// TIA Portal V17 export
// export: Created 2024-08-07T21:44:04.3800599Z, ExportSetting WithDefaults, DisplayName Totally Integrated Automation Portal, DisplayVersion V17 Update 7, DisplayName TIA Portal Openness, DisplayVersion V17 Update 7, DisplayName TIA Portal Version Control Interface, DisplayVersion V17, DisplayName SINAMICS Startdrive Advanced, DisplayVersion V17 SP2, DisplayName SINAMICS Startdrive G110M, G120, G120C, G120D, G120P, G115D, DisplayVersion V17 SP2, DisplayName SINAMICS Startdrive G130, G150, S120, S150, SINAMICS MV, S210, DisplayVersion V17 SP2, DisplayName STEP 7 Professional, DisplayVersion V17 Update 7, DisplayName STEP 7 Safety, DisplayVersion V17 Update 6, DisplayName WinCC Advanced / Unified PC, DisplayVersion V17 Update 7
DATA_BLOCK "CycleTimeMeas_Fitting1_DB"   // DB31
VERSION : 0.1
// stored: AutoNumber true, DBAccessibleFromOPCUA true, DBAccessibleFromWebserver true, InstanceOfName CycleTimeMeas, InstanceOfType FB
"CycleTimeMeas"
   // VAR_INPUT
   //    StartCycle : Bool := FALSE;
   //    ResetHistory : Bool := FALSE;
   // END_VAR
   // VAR
   //    ActualTime : Time := T#0MS;
   //    LastTime : Time := T#12S_830MS;
   //    edge2 : Bool := FALSE;
   //    edge1 : Bool := FALSE;
   //    Suma : DInt := 35860;
   //    Count : DInt := 3;
   //    Max : Time := T#13S_176MS;
   //    Min : Time := T#9S_854MS;
   //    Average : Time := T#11S_953MS;
   //    IEC_Timer_0_Instance { S7_SetPoint := 'True'} : TON_TIME;
   //    History : Array[1..20] of Time;
   //    NewTime : Bool := FALSE;
   // END_VAR
BEGIN
   IEC_Timer_0_Instance.PT := T#8M_20S;
   IEC_Timer_0_Instance.IN := FALSE;
   History[1] := T#12S_830MS;
   History[2] := T#13S_176MS;
   History[3] := T#9S_854MS;
   History[4..20] := T#0MS;
END_DATA_BLOCK
